Universal Robots PolyScope program: UniveralRobots.urp

Program MainProg (createdIn=3.0.0 lastSavedIn=3.0.0 directory=/programs installation=default)
Robot Program (runOnlyOnce=true motionType=MoveJ speed=1.047198 acceleration=1.396263 useActiveTCP=false)
  'Program generated by RoboDK v3.8.4 for UR10 on 17/07/2019 15:17:38'
  'Using nominal kinematics.'
  Call ApproachMove
  Call SprayOn
  Call PaintTop
  Call SprayOn
  Call Retract
SubProgram -> ApproachMove
SubProgram -> SprayOn
SubProgram -> PaintTop
SubProgram -> Retract
SubProgram ApproachMove (keepSynchronizedWithDisk=true trackProgramExecution=false) programFile=/programs/ApproachMove.urp
SubProgram SprayOn (keepSynchronizedWithDisk=true trackProgramExecution=false) programFile=/programs/SprayOn.urp
SubProgram PaintTop (keepSynchronizedWithDisk=true trackProgramExecution=false) programFile=/programs/PaintTop.urp
SubProgram Retract (keepSynchronizedWithDisk=true trackProgramExecution=false) programFile=/programs/Retract.urp
